INTERFACE I_ModbusSlaveRtu EXTENDS I_UniversalModbusSlave

PROPERTY ModbusErrorID : MODBUS_ERRORS
GET
END_GET
SET
END_SET
END_PROPERTY

END_INTERFACE

(* stored: Version 1.1.0.1, ProductVersion 3.1.4024.12
   Itf I_ModbusSlaveRtu: Id {f6cc8562-becd-4eee-9889-c7c39fc121d0}
   Property ModbusErrorID: Id {104d4279-78f3-4a2b-abfb-5f74257f2b8a}
   Get Get: Id {c488a572-8a84-4064-b5dc-1c1f779e9737}
   Set Set: Id {44a6c67d-c825-46fe-ae17-ba209b391519} *)
